(* Logix 5000 project; controller PLC_L27ERM_QBFC1B vendor 1 type 14 code 151 rev 33.13; software revision 33.01 *)

TASK MainTask (continuous, watchdog 500 ms) : MainProgram, CF

MODULES
   Local : vendor 1 type 14 code 151 (Compact 0, rev 33.13)
      Counters : Embedded (Compact 3, rev 1.1, Output RPI 20 ms)
      Discrete_IO : Embedded (Compact 1, rev 3.1, Output RPI 20 ms)
      Analog_IO : Embedded (Compact 2, rev 1.1, Output RPI 80 ms)
      PowerFlex755 : vendor 1 type 143 code 6288 (Ethernet 192.168.2.10, rev 3.2, Output RPI 20 ms)
          : vendor 1 type 143 code 416 (RhinoBP 5, rev 1.8)
          : vendor 1 type 143 code 416 (RhinoBP 4, rev 1.8)
          : vendor 1 type 143 code 32928 (RhinoBP 13, rev 1.1)
          : vendor 1 type 143 code 416 (RhinoBP 6, rev 1.8)
          : vendor 1 type 143 code 33184 (RhinoBP 14, rev 2.5)
END_MODULES

TYPE AnlgIn :
STRUCT
   SCALE_CH : SCALE[4];
   Selector_CH : INT[4];
   PresionEntrada : REAL;
   PresionDescarga : REAL;
   TemperaturaEntrada : REAL;
   TemperaturaDescarga : REAL;
   TemperaturaMotor : REAL;
   PresionCasing : REAL;
   PresionTHP : REAL;
   TemperaturaTHT : REAL;
   ReferenciaAnlg : REAL;
   CTTransformadorElevador : REAL;
   Vibration : REAL;
   CorrienteFuga : REAL;
END_STRUCT
END_TYPE

TYPE DHS :   // Datos sensor de fondo
STRUCT
   PresionEntrada : REAL;
   PresionDescarga : REAL;
   TemperaturaEntrada : REAL;
   TemperaturaDescarga : REAL;
   TemperaturaMotor : REAL;
   PresionCasing : REAL;
   PresionTHP : REAL;
   TemperaturaTHT : REAL;
   Fuente : BOOL;
   Vibration : REAL;
   CorrienteFuga : REAL;
END_STRUCT
END_TYPE

TYPE DInput :   // Fn. Entrada digital
STRUCT
   Start : BMUX;   // Arranque
   Stop : BMUX;   // Parada
   Reset : BMUX;   // Reset
   StopESD : BMUX;   // ESD
   DisparoAltoNivelAceiteSUT : BMUX;   // Disparo SUT
   DisparoAltaTemperaturaSUT : BMUX;   // Disparo SUT
   AlarmaAltaTemperaturaSUT : BMUX;   // Alarma SUT
   AlarmaBajoNivelAceiteSUT : BMUX;   // Alarma SUT
   DisparoBajoBajoNivelAceiteSUT : BMUX;   // Disparo SUT
   DisparoValvulaSobrePresionSUT : BMUX;   // Disparo SUT
   DisparoSobreTensionSUT : BMUX;   // Disparo Tension
   AlarmaDPS : BMUX;   // Alarma DPS
   DisparoAltaTemperaturaFiltros : BMUX;   // Disparo Filtros
   DisparoAltaPresionTHP : BMUX;   // Disparo Instrumentación
   DisparoAltaTemperaturaTHT : BMUX;   // Disparo Instrumentación
   StopESDRemoto : BMUX;   // ESD Remoto
   DisparoPuertaAbierta : BMUX;   // Disparo CILA2S
   DisparoTermicoMotor : BMUX;   // Disparo Motor
   DisparoShutdownSCC : BMUX;   // Disparo SCC
   DisparoBajaPresionTroncal : BMUX;   // Disparo SCC
END_STRUCT
END_TYPE

TYPE DOutput :   // Salida digital
STRUCT
   DO0 : BMUX;
   DO1 : BMUX;
   DO2 : BMUX;
   DO3 : BMUX;
   DO4 : BMUX;
   DO5 : BMUX;
   DO6 : BMUX;
   DO7 : BMUX;
END_STRUCT
END_TYPE

TYPE Filtro :   // Filtro armónicos
STRUCT
   Valor : REAL;
   Referencia : REAL;
   TiempoMuerto : TIMER;
   Output : BOOL;
END_STRUCT
END_TYPE

TYPE IOFn :   // Fn. Salida digital
STRUCT
   DisparoBreakerESD : BOOL;
   FiltroArmonicos : BOOL;
   FallaGeneral : BOOL;
   EstadoCILA2S : BOOL;   // 1:Activo 0:Detenido
   IOFnWord : INT;
END_STRUCT
END_TYPE

ADD_ON_INSTRUCTION BMUX   (* revision 1.1 Multiplexor, vendor Jorge Alberto MartÃ­nez SuÃ¡rez *)
// Multiplexor digital 16:1
// Revision note:
// Se contemplan entradas NO y NC
VAR_INPUT
   Input : INT; {visible}   // Entrada MUX
END_VAR
VAR_OUTPUT
   Output : BOOL; {visible}   // Salida MUX
END_VAR
VAR_INPUT
   Selector : INT; {visible}   // Selector MUX
   Type : BOOL; {visible}
END_VAR

ROUTINE Logic   (* structured text *)
   // Case para las entradas del Add-On
   case Selector of
   	0: 	Output 	:= 0;
   	1: 	Output 	:= Input.0;
   	2: 	Output 	:= Input.1;
   	3: 	Output 	:= Input.2;
   	4: 	Output 	:= Input.3;
   	5: 	Output 	:= Input.4;
   	6: 	Output 	:= Input.5;
   	7: 	Output 	:= Input.6;
   	8: 	Output 	:= Input.7;
   	9: 	Output 	:= Input.8;
   	10: Output 	:= Input.9;
   	11: Output 	:= Input.10;
   	12: Output 	:= Input.11;
   	13: Output 	:= Input.12;
   	14: Output 	:= Input.13;
   	15: Output 	:= Input.14;
   	16: Output	:= Input.15;
   	else
   		Output 	:= 0;
   end_case;
   
   // Tipo de entrada 0:NO 1:NC
   if Type then
   	Output := NOT Output;
   end_if;
   
   // Deshabilitar Salida del Add-On
   if NOT EnableIn then
   	Output := 0;
   end_if;
END_ROUTINE
END_ADD_ON_INSTRUCTION

VAR_GLOBAL   (* controller tags *)
   EstadoDrive : BOOL;
   RelTX : REAL := 1.0;
   Reset : BOOL;
   TensionEntrada : REAL;
END_VAR

PROGRAM CF   (* main routine MainRoutineCF *)
VAR
   AtSetpointSPD : BOOL;
   MtrSpd : REAL;
   PR_E : INT;
   PRDHz : REAL;
   PRH : REAL;
   PRHMS : REAL;
   PRHz : REAL;
   PRM : REAL;
   PRS : REAL;
   RefNotReached : BOOL;
   RefReached : BOOL;
   Rtrn : REAL;
   Start : BOOL;
END_VAR

ROUTINE MainRoutineCF   (* ladder *)
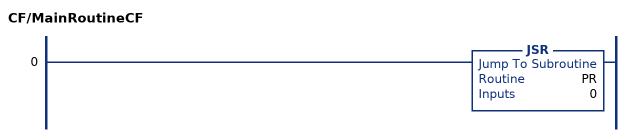
   0: JSR(PR,0);
END_ROUTINE

ROUTINE PR   (* structured text *)
   // LÓGICA SECUENCIAL
   // E0 -> E1
   if PR_E.0 AND Start then
   	PR_E.1:=1; PR_E.0:=0;
   end_if;
   
   // E1 -> E2
   if PR_E.1 AND AtSetpointSPD then
   	PR_E.2:=1; PR_E.1:=0;
   end_if;
   
   // E2 -> E1
   if PR_E.2 AND RefNotReached then
   	PR_E.1:=1; PR_E.2:=0;
   end_if;
   
   // E2 -> E0
   if PR_E.2 AND RefReached then
   	PR_E.0:=1; PR_E.2:=0;
   end_if;
   
   // LÓGICA COMBINACIONAL
   // Estado 0
   if PR_E.0 then
   	PRHMS:= PRH*3600 + PRM*60 + PRS;
   end_if;
   
   // Estado 1
   if PR_E.1 & (PRHz < MtrSpd) then
   	Rtrn := MtrSpd - PRDHz;
   end_if;
   
   if PR_E.1 & (PRHz > MtrSpd) then
   	Rtrn := MtrSpd + PRDHz;
   end_if;
END_ROUTINE
END_PROGRAM

PROGRAM MainProgram   (* main routine MainRoutine *)
VAR
   AnlgFn : AnlgIn;
   CorrienteMotor : REAL;
   DInput : DInput := (Start.Selector := 1, Stop.Selector := 2, Reset.Selector := 3);
   DOutput : DOutput := (DO0.Selector := 4);
   HF : Filtro := (Referencia := 100.0, TiempoMuerto.PRE := 10000);
   index : INT;
   IOFn : IOFn;
        .IOFnWord.0   // Falla general
        .IOFnWord.1   // Disparo breaker ESD
        .IOFnWord.2   // Filtro de armónicos
        .IOFnWord.3   // Estado CILA2S (Activo/Detenido)
   ParadaProteccion : INT;   // Lista de paradas por protección
        .0   // Parada por Presión de entrada
        .1   // Parada por presión de descarga
        .10   // Parada por BUS DC
        .11   // Parada por corriente de salida VSD
        .12   // Parada por tensión de entrada
        .13   // Parada por corriente de motor
        .2   // Parada por temperatura de entrada
        .3   // Parada por temperatura de descarga
        .4   // Parada por temperatura de motor
        .5   // Parada por presión de casing
        .6   // Parada por presión THP
        .7   // Parada por temperatura THT
        .8   // Parada por Vibración
        .9   // Parada por corriente de fuga
   ProtBusDC : ALARM_ANALOG;
   ProtCorrienteFuga : ALARM_ANALOG;
   ProtCorrienteMotor : ALARM_ANALOG;
   ProtOutputCurrent : ALARM_ANALOG;
   ProtPresionCasing : ALARM_ANALOG;
   ProtPresionDescarga : ALARM_ANALOG;
   ProtPresionEntrada : ALARM_ANALOG;
   ProtPresionTHP : ALARM_ANALOG;
   ProtStopVSD : INT;
   ProtTemperaturaDescarga : ALARM_ANALOG;
   ProtTemperaturaEntrada : ALARM_ANALOG;
   ProtTemperaturaMotor : ALARM_ANALOG;
   ProtTemperaturaTHT : ALARM_ANALOG;
   ProtTensionEntrada : ALARM_ANALOG;
   ProtVibration : ALARM_ANALOG;
   SensorFondo : DHS;
END_VAR

ROUTINE AnlgIn   (* structured text *)
   // Escalizar todos los canales
   AnlgFn.SCALE_CH[0].In := Local:2:I.Ch0Data;
   AnlgFn.SCALE_CH[1].In := Local:2:I.Ch1Data;
   AnlgFn.SCALE_CH[2].In := Local:2:I.Ch2Data;
   AnlgFn.SCALE_CH[3].In := Local:2:I.Ch3Data;
   
   // For para asignar las variables de proceso
   for index:=0 to 3 do
   	case AnlgFn.Selector_CH[index] of
   	1: AnlgFn.PresionEntrada := AnlgFn.SCALE_CH[index].Out;
   	2: AnlgFn.PresionDescarga:= AnlgFn.SCALE_CH[index].Out;
   	3: AnlgFn.TemperaturaEntrada := AnlgFn.SCALE_CH[index].Out;
   	4: AnlgFn.TemperaturaDescarga:= AnlgFn.SCALE_CH[index].Out;
   	5: AnlgFn.TemperaturaMotor:= AnlgFn.SCALE_CH[index].Out;
   	6: AnlgFn.PresionCasing:= AnlgFn.SCALE_CH[index].Out;
   	7: AnlgFn.PresionTHP:= AnlgFn.SCALE_CH[index].Out;
   	8: AnlgFn.TemperaturaTHT:= AnlgFn.SCALE_CH[index].Out;
   	9: AnlgFn.ReferenciaAnlg:= AnlgFn.SCALE_CH[index].Out;
   	10: AnlgFn.CTTransformadorElevador:= AnlgFn.SCALE_CH[index].Out;
   	11: AnlgFn.Vibration:= AnlgFn.SCALE_CH[index].Out;
   	12: AnlgFn.CorrienteFuga:= AnlgFn.SCALE_CH[index].Out;
   
   	end_case;
   end_for;
END_ROUTINE

ROUTINE DigitalFn   (* ladder *)
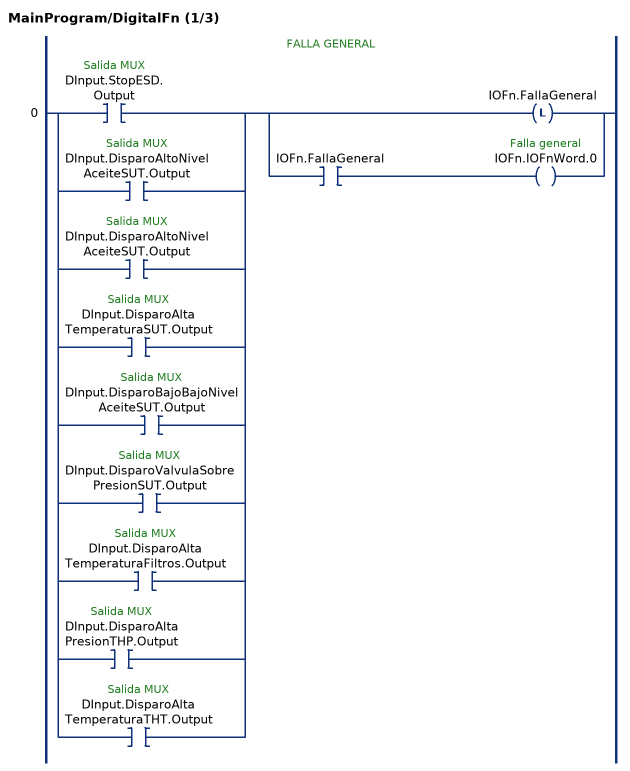
   // FALLA GENERAL
   0: [XIC(DInput.StopESD.Output) ,XIC(DInput.DisparoAltoNivelAceiteSUT.Output) ,XIC(DInput.DisparoAltoNivelAceiteSUT.Output) ,XIC(DInput.DisparoAltaTemperaturaSUT.Output) ,XIC(DInput.DisparoBajoBajoNivelAceiteSUT.Output) ,XIC(DInput.DisparoValvulaSobrePresionSUT.Output) ,XIC(DInput.DisparoAltaTemperaturaFiltros.Output) ,XIC(DInput.DisparoAltaPresionTHP.Output) ,XIC(DInput.DisparoAltaTemperaturaTHT.Output) ][OTL(IOFn.FallaGeneral) ,XIC(IOFn.FallaGeneral) OTE(IOFn.IOFnWord.0) ];
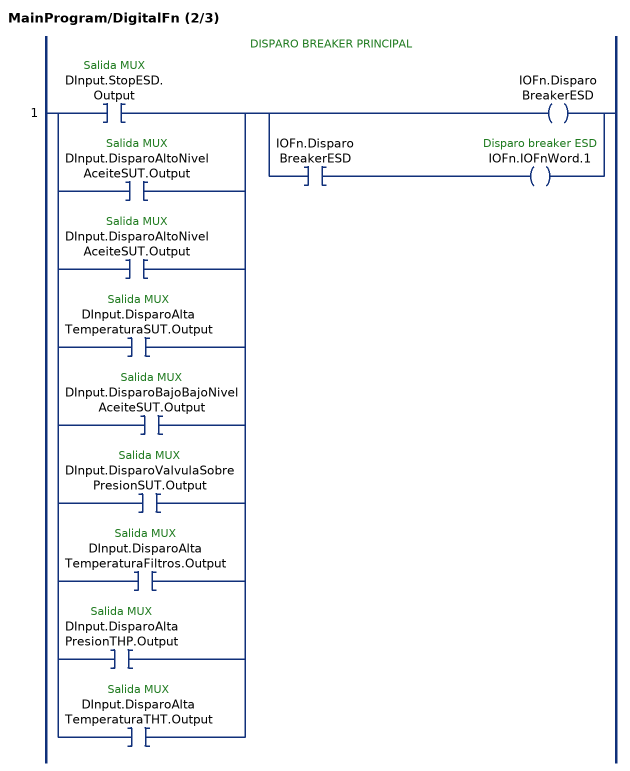
   // DISPARO BREAKER PRINCIPAL
   1: [XIC(DInput.StopESD.Output) ,XIC(DInput.DisparoAltoNivelAceiteSUT.Output) ,XIC(DInput.DisparoAltoNivelAceiteSUT.Output) ,XIC(DInput.DisparoAltaTemperaturaSUT.Output) ,XIC(DInput.DisparoBajoBajoNivelAceiteSUT.Output) ,XIC(DInput.DisparoValvulaSobrePresionSUT.Output) ,XIC(DInput.DisparoAltaTemperaturaFiltros.Output) ,XIC(DInput.DisparoAltaPresionTHP.Output) ,XIC(DInput.DisparoAltaTemperaturaTHT.Output) ][OTE(IOFn.DisparoBreakerESD) ,XIC(IOFn.DisparoBreakerESD) OTE(IOFn.IOFnWord.1) ];
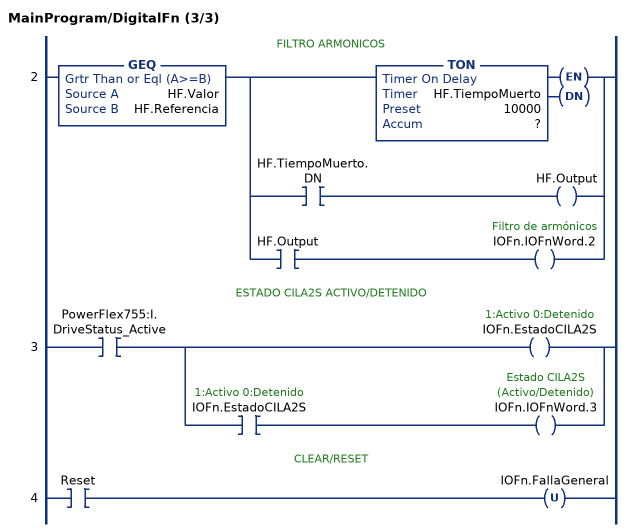
   // FILTRO ARMONICOS
   2: GEQ(HF.Valor,HF.Referencia)[TON(HF.TiempoMuerto,?,?) ,XIC(HF.TiempoMuerto.DN) OTE(HF.Output) ,XIC(HF.Output) OTE(IOFn.IOFnWord.2) ];
   // ESTADO CILA2S ACTIVO/DETENIDO
   3: XIC(PowerFlex755:I.DriveStatus_Active)[OTE(IOFn.EstadoCILA2S) ,XIC(IOFn.EstadoCILA2S) OTE(IOFn.IOFnWord.3) ];
   // CLEAR/RESET
   4: XIC(Reset)OTU(IOFn.FallaGeneral);
END_ROUTINE

ROUTINE InputLD   (* ladder *)
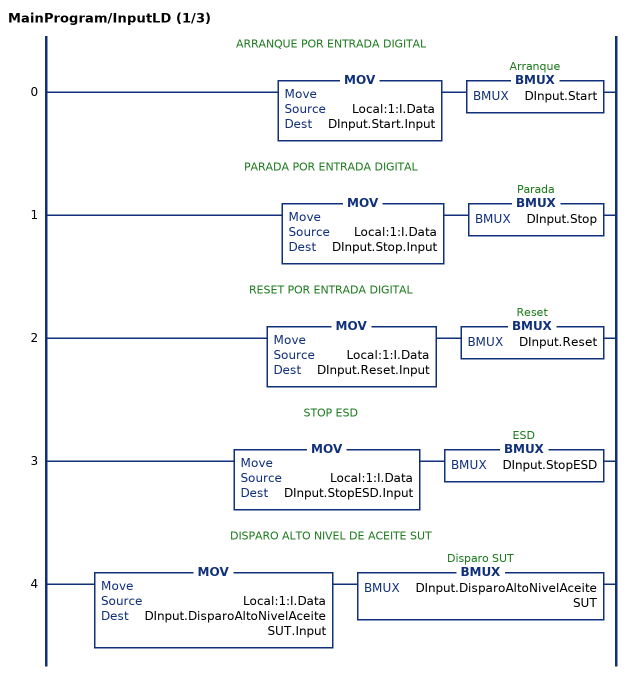
   // ARRANQUE POR ENTRADA DIGITAL
   0: MOV(Local:1:I.Data,DInput.Start.Input)BMUX(DInput.Start);
   // PARADA POR ENTRADA DIGITAL
   1: MOV(Local:1:I.Data,DInput.Stop.Input)BMUX(DInput.Stop);
   // RESET POR ENTRADA DIGITAL
   2: MOV(Local:1:I.Data,DInput.Reset.Input)BMUX(DInput.Reset);
   // STOP ESD
   3: MOV(Local:1:I.Data,DInput.StopESD.Input)BMUX(DInput.StopESD);
   // DISPARO ALTO NIVEL DE ACEITE SUT
   4: MOV(Local:1:I.Data,DInput.DisparoAltoNivelAceiteSUT.Input)BMUX(DInput.DisparoAltoNivelAceiteSUT);
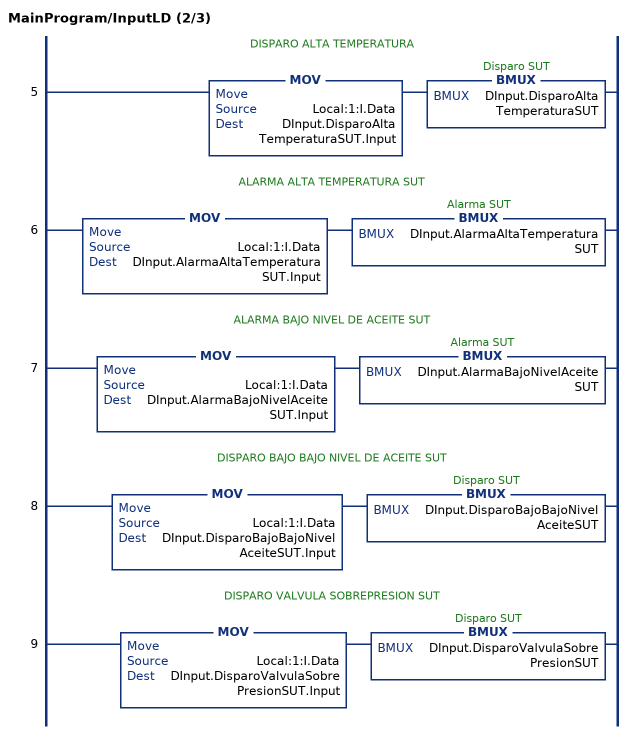
   // DISPARO ALTA TEMPERATURA
   5: MOV(Local:1:I.Data,DInput.DisparoAltaTemperaturaSUT.Input)BMUX(DInput.DisparoAltaTemperaturaSUT);
   // ALARMA ALTA TEMPERATURA SUT
   6: MOV(Local:1:I.Data,DInput.AlarmaAltaTemperaturaSUT.Input)BMUX(DInput.AlarmaAltaTemperaturaSUT);
   // ALARMA BAJO NIVEL DE ACEITE SUT
   7: MOV(Local:1:I.Data,DInput.AlarmaBajoNivelAceiteSUT.Input)BMUX(DInput.AlarmaBajoNivelAceiteSUT);
   // DISPARO BAJO BAJO NIVEL DE ACEITE SUT
   8: MOV(Local:1:I.Data,DInput.DisparoBajoBajoNivelAceiteSUT.Input)BMUX(DInput.DisparoBajoBajoNivelAceiteSUT);
   // DISPARO VALVULA SOBREPRESION SUT
   9: MOV(Local:1:I.Data,DInput.DisparoValvulaSobrePresionSUT.Input)BMUX(DInput.DisparoValvulaSobrePresionSUT);
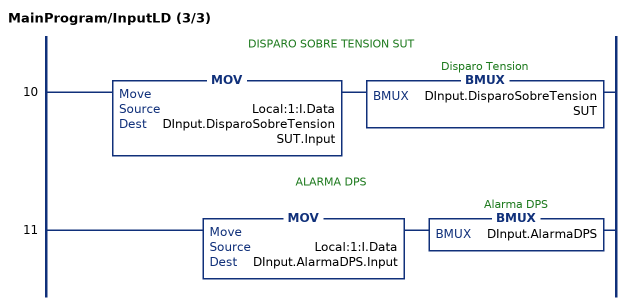
   // DISPARO SOBRE TENSION SUT
   10: MOV(Local:1:I.Data,DInput.DisparoSobreTensionSUT.Input)BMUX(DInput.DisparoSobreTensionSUT);
   // ALARMA DPS
   11: MOV(Local:1:I.Data,DInput.AlarmaDPS.Input)BMUX(DInput.AlarmaDPS);
END_ROUTINE

ROUTINE MainRoutine   (* ladder *)
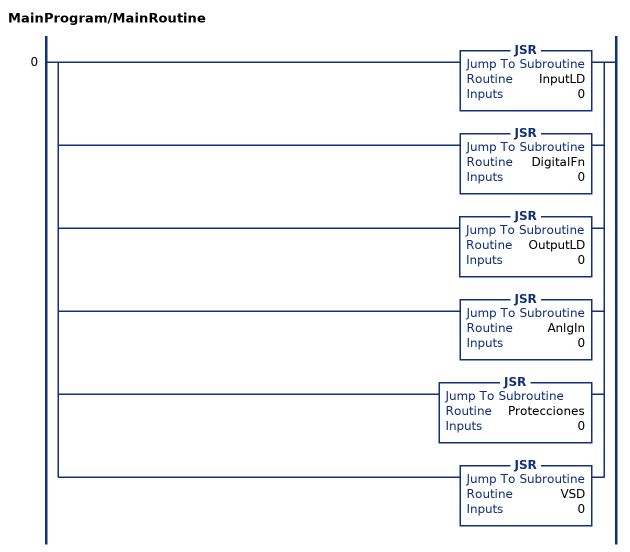
   0: [JSR(InputLD,0) ,JSR(DigitalFn,0) ,JSR(OutputLD,0) ,JSR(AnlgIn,0) ,JSR(Protecciones,0) ,JSR(VSD,0) ];
END_ROUTINE

ROUTINE OutputLD   (* ladder *)
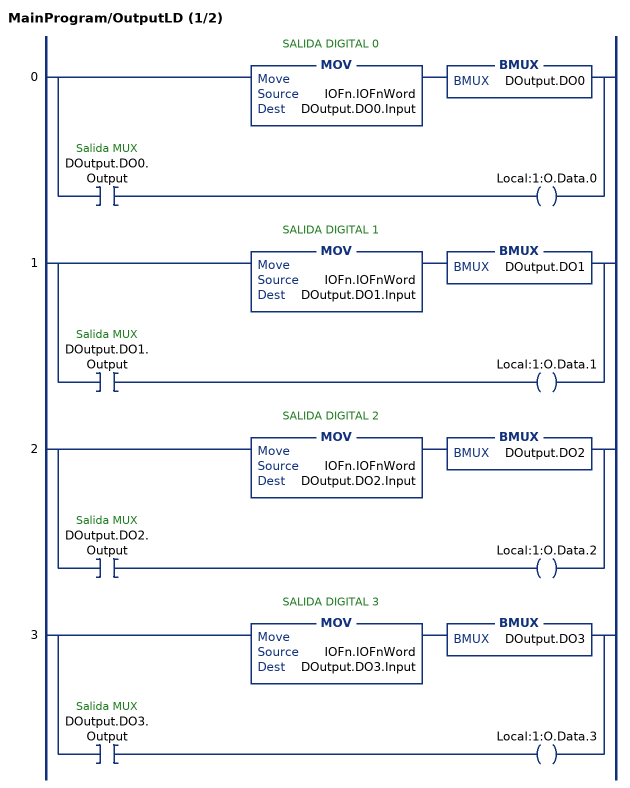
   // SALIDA DIGITAL 0
   0: [MOV(IOFn.IOFnWord,DOutput.DO0.Input) BMUX(DOutput.DO0) ,XIC(DOutput.DO0.Output) OTE(Local:1:O.Data.0) ];
   // SALIDA DIGITAL 1
   1: [MOV(IOFn.IOFnWord,DOutput.DO1.Input) BMUX(DOutput.DO1) ,XIC(DOutput.DO1.Output) OTE(Local:1:O.Data.1) ];
   // SALIDA DIGITAL 2
   2: [MOV(IOFn.IOFnWord,DOutput.DO2.Input) BMUX(DOutput.DO2) ,XIC(DOutput.DO2.Output) OTE(Local:1:O.Data.2) ];
   // SALIDA DIGITAL 3
   3: [MOV(IOFn.IOFnWord,DOutput.DO3.Input) BMUX(DOutput.DO3) ,XIC(DOutput.DO3.Output) OTE(Local:1:O.Data.3) ];
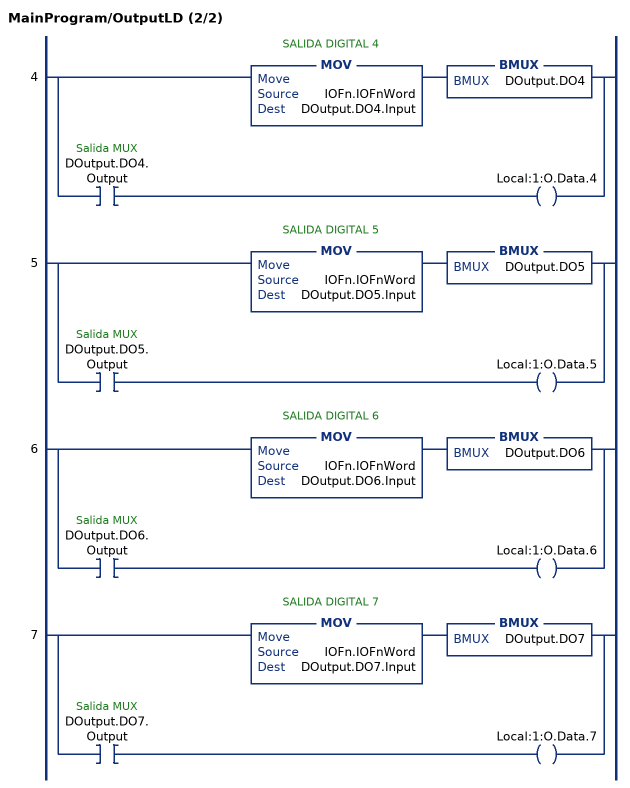
   // SALIDA DIGITAL 4
   4: [MOV(IOFn.IOFnWord,DOutput.DO4.Input) BMUX(DOutput.DO4) ,XIC(DOutput.DO4.Output) OTE(Local:1:O.Data.4) ];
   // SALIDA DIGITAL 5
   5: [MOV(IOFn.IOFnWord,DOutput.DO5.Input) BMUX(DOutput.DO5) ,XIC(DOutput.DO5.Output) OTE(Local:1:O.Data.5) ];
   // SALIDA DIGITAL 6
   6: [MOV(IOFn.IOFnWord,DOutput.DO6.Input) BMUX(DOutput.DO6) ,XIC(DOutput.DO6.Output) OTE(Local:1:O.Data.6) ];
   // SALIDA DIGITAL 7
   7: [MOV(IOFn.IOFnWord,DOutput.DO7.Input) BMUX(DOutput.DO7) ,XIC(DOutput.DO7.Output) OTE(Local:1:O.Data.7) ];
END_ROUTINE

ROUTINE Protecciones   (* ladder *)
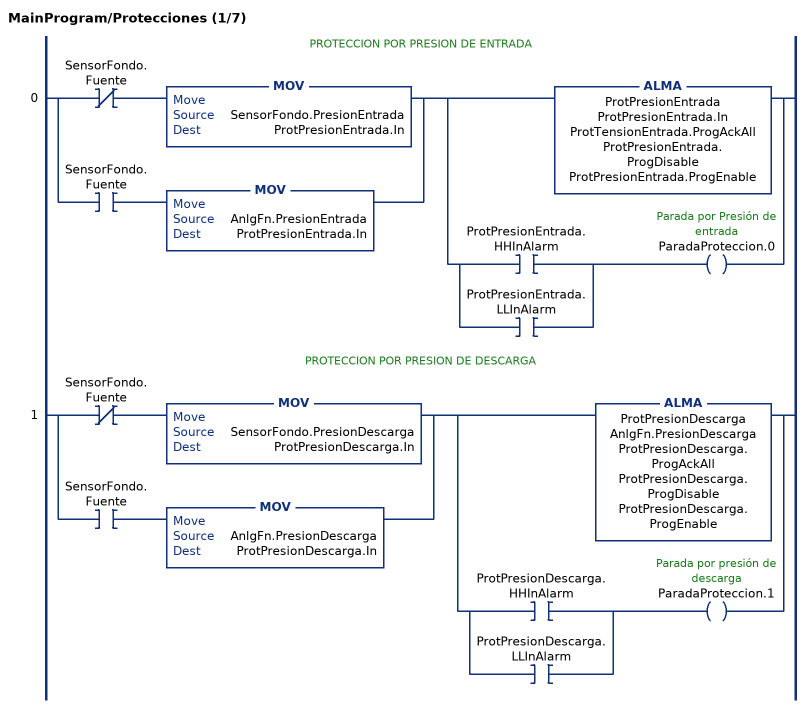
   // PROTECCION POR PRESION DE ENTRADA
   0: [XIO(SensorFondo.Fuente) MOV(SensorFondo.PresionEntrada,ProtPresionEntrada.In) ,XIC(SensorFondo.Fuente) MOV(AnlgFn.PresionEntrada,ProtPresionEntrada.In) ][ALMA(ProtPresionEntrada,ProtPresionEntrada.In,ProtTensionEntrada.ProgAckAll,ProtPresionEntrada.ProgDisable,ProtPresionEntrada.ProgEnable) ,[XIC(ProtPresionEntrada.HHInAlarm) ,XIC(ProtPresionEntrada.LLInAlarm) ] OTE(ParadaProteccion.0) ];
   // PROTECCION POR PRESION DE DESCARGA
   1: [XIO(SensorFondo.Fuente) MOV(SensorFondo.PresionDescarga,ProtPresionDescarga.In) ,XIC(SensorFondo.Fuente) MOV(AnlgFn.PresionDescarga,ProtPresionDescarga.In) ][ALMA(ProtPresionDescarga,AnlgFn.PresionDescarga,ProtPresionDescarga.ProgAckAll,ProtPresionDescarga.ProgDisable,ProtPresionDescarga.ProgEnable) ,[XIC(ProtPresionDescarga.HHInAlarm) ,XIC(ProtPresionDescarga.LLInAlarm) ] OTE(ParadaProteccion.1) ];
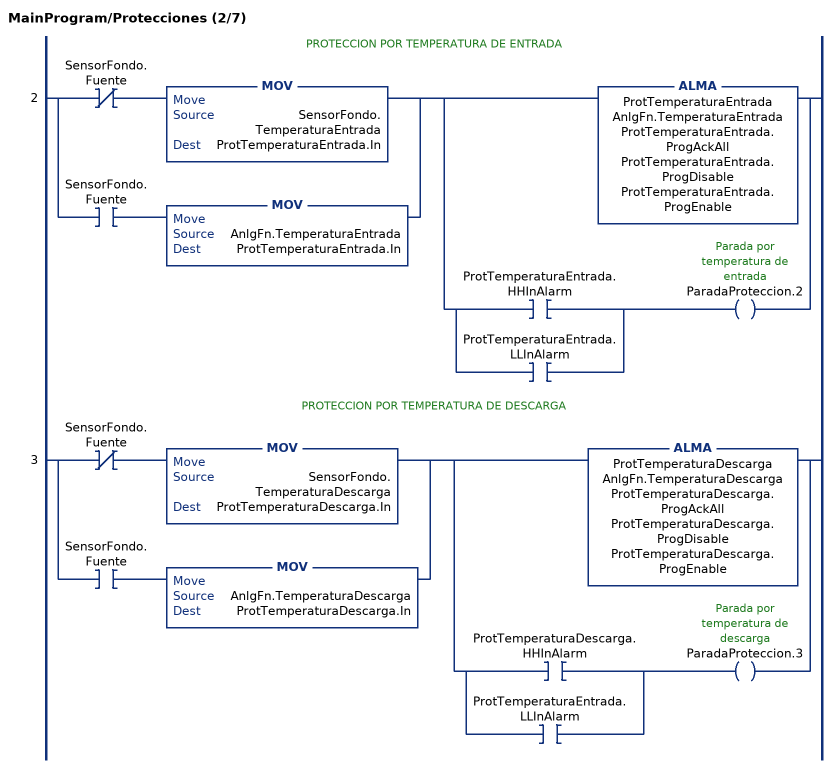
   // PROTECCION POR TEMPERATURA DE ENTRADA
   2: [XIO(SensorFondo.Fuente) MOV(SensorFondo.TemperaturaEntrada,ProtTemperaturaEntrada.In) ,XIC(SensorFondo.Fuente) MOV(AnlgFn.TemperaturaEntrada,ProtTemperaturaEntrada.In) ][ALMA(ProtTemperaturaEntrada,AnlgFn.TemperaturaEntrada,ProtTemperaturaEntrada.ProgAckAll,ProtTemperaturaEntrada.ProgDisable,ProtTemperaturaEntrada.ProgEnable) ,[XIC(ProtTemperaturaEntrada.HHInAlarm) ,XIC(ProtTemperaturaEntrada.LLInAlarm) ] OTE(ParadaProteccion.2) ];
   // PROTECCION POR TEMPERATURA DE DESCARGA
   3: [XIO(SensorFondo.Fuente) MOV(SensorFondo.TemperaturaDescarga,ProtTemperaturaDescarga.In) ,XIC(SensorFondo.Fuente) MOV(AnlgFn.TemperaturaDescarga,ProtTemperaturaDescarga.In) ][ALMA(ProtTemperaturaDescarga,AnlgFn.TemperaturaDescarga,ProtTemperaturaDescarga.ProgAckAll,ProtTemperaturaDescarga.ProgDisable,ProtTemperaturaDescarga.ProgEnable) ,[XIC(ProtTemperaturaDescarga.HHInAlarm) ,XIC(ProtTemperaturaEntrada.LLInAlarm) ] OTE(ParadaProteccion.3) ];
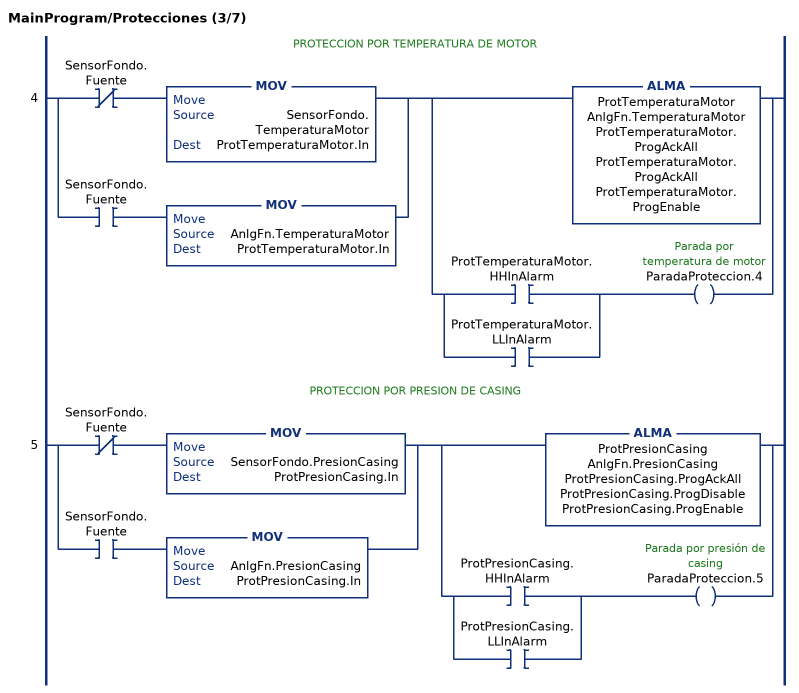
   // PROTECCION POR TEMPERATURA DE MOTOR
   4: [XIO(SensorFondo.Fuente) MOV(SensorFondo.TemperaturaMotor,ProtTemperaturaMotor.In) ,XIC(SensorFondo.Fuente) MOV(AnlgFn.TemperaturaMotor,ProtTemperaturaMotor.In) ][ALMA(ProtTemperaturaMotor,AnlgFn.TemperaturaMotor,ProtTemperaturaMotor.ProgAckAll,ProtTemperaturaMotor.ProgAckAll,ProtTemperaturaMotor.ProgEnable) ,[XIC(ProtTemperaturaMotor.HHInAlarm) ,XIC(ProtTemperaturaMotor.LLInAlarm) ] OTE(ParadaProteccion.4) ];
   // PROTECCION POR PRESION DE CASING
   5: [XIO(SensorFondo.Fuente) MOV(SensorFondo.PresionCasing,ProtPresionCasing.In) ,XIC(SensorFondo.Fuente) MOV(AnlgFn.PresionCasing,ProtPresionCasing.In) ][ALMA(ProtPresionCasing,AnlgFn.PresionCasing,ProtPresionCasing.ProgAckAll,ProtPresionCasing.ProgDisable,ProtPresionCasing.ProgEnable) ,[XIC(ProtPresionCasing.HHInAlarm) ,XIC(ProtPresionCasing.LLInAlarm) ] OTE(ParadaProteccion.5) ];
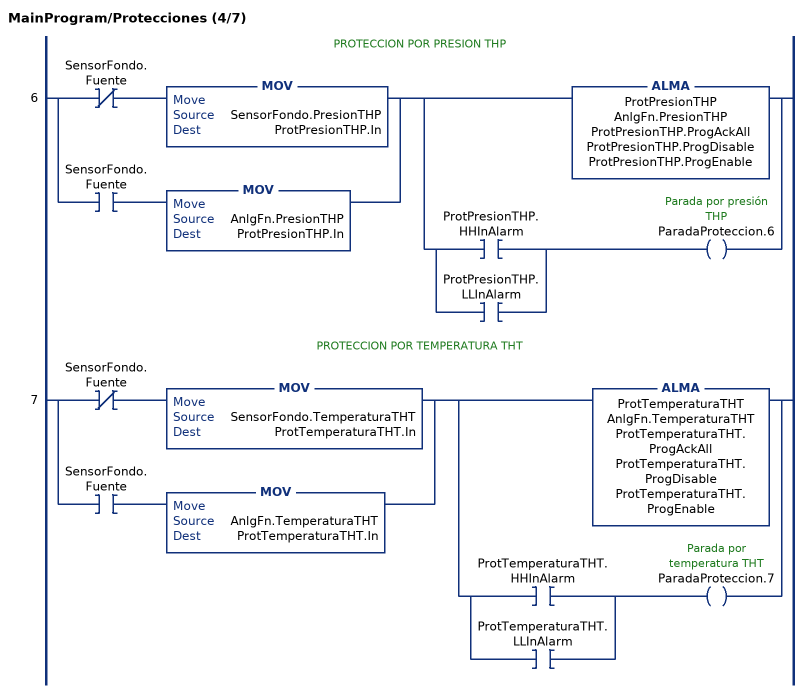
   // PROTECCION POR PRESION THP
   6: [XIO(SensorFondo.Fuente) MOV(SensorFondo.PresionTHP,ProtPresionTHP.In) ,XIC(SensorFondo.Fuente) MOV(AnlgFn.PresionTHP,ProtPresionTHP.In) ][ALMA(ProtPresionTHP,AnlgFn.PresionTHP,ProtPresionTHP.ProgAckAll,ProtPresionTHP.ProgDisable,ProtPresionTHP.ProgEnable) ,[XIC(ProtPresionTHP.HHInAlarm) ,XIC(ProtPresionTHP.LLInAlarm) ] OTE(ParadaProteccion.6) ];
   // PROTECCION POR TEMPERATURA THT
   7: [XIO(SensorFondo.Fuente) MOV(SensorFondo.TemperaturaTHT,ProtTemperaturaTHT.In) ,XIC(SensorFondo.Fuente) MOV(AnlgFn.TemperaturaTHT,ProtTemperaturaTHT.In) ][ALMA(ProtTemperaturaTHT,AnlgFn.TemperaturaTHT,ProtTemperaturaTHT.ProgAckAll,ProtTemperaturaTHT.ProgDisable,ProtTemperaturaTHT.ProgEnable) ,[XIC(ProtTemperaturaTHT.HHInAlarm) ,XIC(ProtTemperaturaTHT.LLInAlarm) ] OTE(ParadaProteccion.7) ];
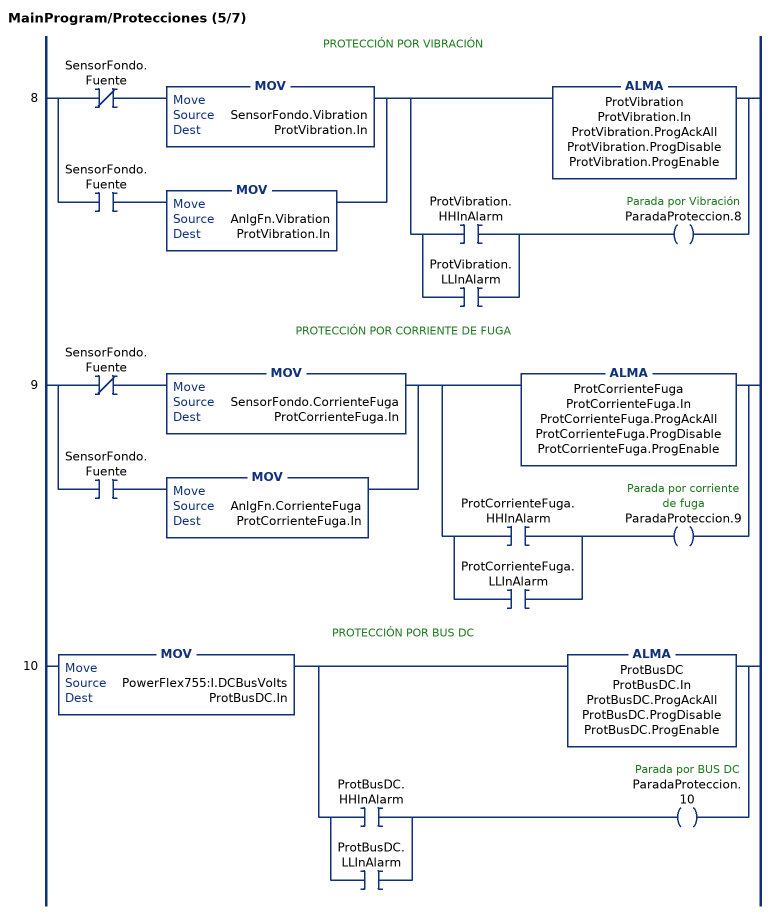
   // PROTECCIÓN POR VIBRACIÓN
   8: [XIO(SensorFondo.Fuente) MOV(SensorFondo.Vibration,ProtVibration.In) ,XIC(SensorFondo.Fuente) MOV(AnlgFn.Vibration,ProtVibration.In) ][ALMA(ProtVibration,ProtVibration.In,ProtVibration.ProgAckAll,ProtVibration.ProgDisable,ProtVibration.ProgEnable) ,[XIC(ProtVibration.HHInAlarm) ,XIC(ProtVibration.LLInAlarm) ] OTE(ParadaProteccion.8) ];
   // PROTECCIÓN POR CORRIENTE DE FUGA
   9: [XIO(SensorFondo.Fuente) MOV(SensorFondo.CorrienteFuga,ProtCorrienteFuga.In) ,XIC(SensorFondo.Fuente) MOV(AnlgFn.CorrienteFuga,ProtCorrienteFuga.In) ][ALMA(ProtCorrienteFuga,ProtCorrienteFuga.In,ProtCorrienteFuga.ProgAckAll,ProtCorrienteFuga.ProgDisable,ProtCorrienteFuga.ProgEnable) ,[XIC(ProtCorrienteFuga.HHInAlarm) ,XIC(ProtCorrienteFuga.LLInAlarm) ] OTE(ParadaProteccion.9) ];
   // PROTECCIÓN POR BUS DC
   10: MOV(PowerFlex755:I.DCBusVolts,ProtBusDC.In)[ALMA(ProtBusDC,ProtBusDC.In,ProtBusDC.ProgAckAll,ProtBusDC.ProgDisable,ProtBusDC.ProgEnable) ,[XIC(ProtBusDC.HHInAlarm) ,XIC(ProtBusDC.LLInAlarm) ] OTE(ParadaProteccion.10) ];
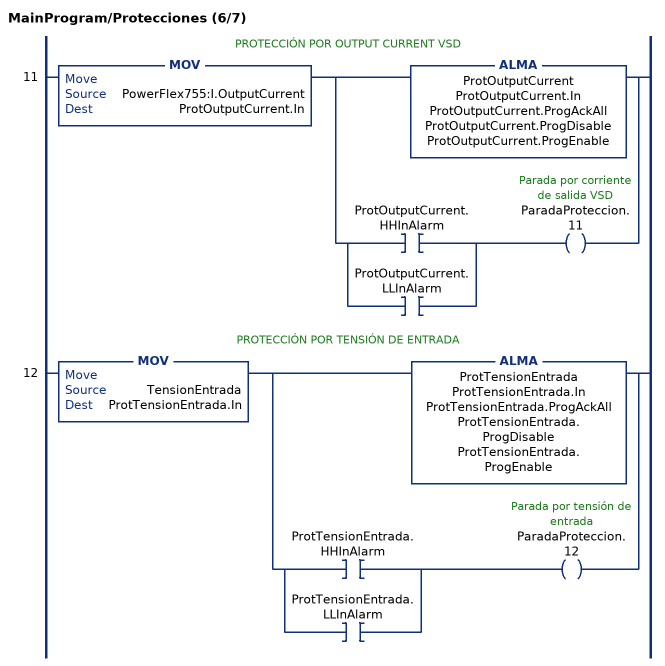
   // PROTECCIÓN POR OUTPUT CURRENT VSD
   11: MOV(PowerFlex755:I.OutputCurrent,ProtOutputCurrent.In)[ALMA(ProtOutputCurrent,ProtOutputCurrent.In,ProtOutputCurrent.ProgAckAll,ProtOutputCurrent.ProgDisable,ProtOutputCurrent.ProgEnable) ,[XIC(ProtOutputCurrent.HHInAlarm) ,XIC(ProtOutputCurrent.LLInAlarm) ] OTE(ParadaProteccion.11) ];
   // PROTECCIÓN POR TENSIÓN DE ENTRADA
   12: MOV(TensionEntrada,ProtTensionEntrada.In)[ALMA(ProtTensionEntrada,ProtTensionEntrada.In,ProtTensionEntrada.ProgAckAll,ProtTensionEntrada.ProgDisable,ProtTensionEntrada.ProgEnable) ,[XIC(ProtTensionEntrada.HHInAlarm) ,XIC(ProtTensionEntrada.LLInAlarm) ] OTE(ParadaProteccion.12) ];
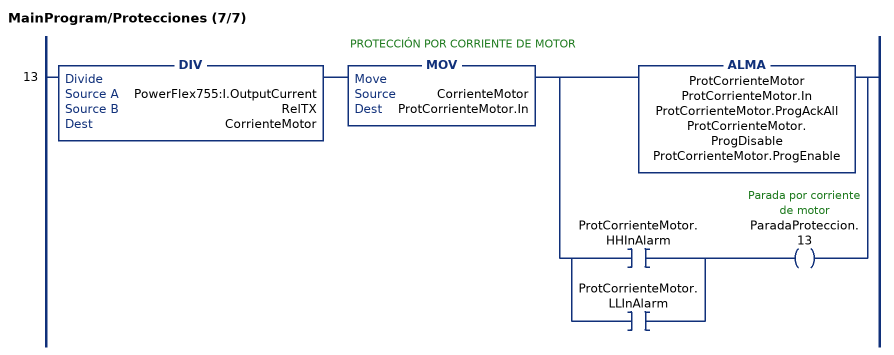
   // PROTECCIÓN POR CORRIENTE DE MOTOR
   13: DIV(PowerFlex755:I.OutputCurrent,RelTX,CorrienteMotor)MOV(CorrienteMotor,ProtCorrienteMotor.In)[ALMA(ProtCorrienteMotor,ProtCorrienteMotor.In,ProtCorrienteMotor.ProgAckAll,ProtCorrienteMotor.ProgDisable,ProtCorrienteMotor.ProgEnable) ,[XIC(ProtCorrienteMotor.HHInAlarm) ,XIC(ProtCorrienteMotor.LLInAlarm) ] OTE(ParadaProteccion.13) ];
END_ROUTINE

ROUTINE VSD   (* ladder *)
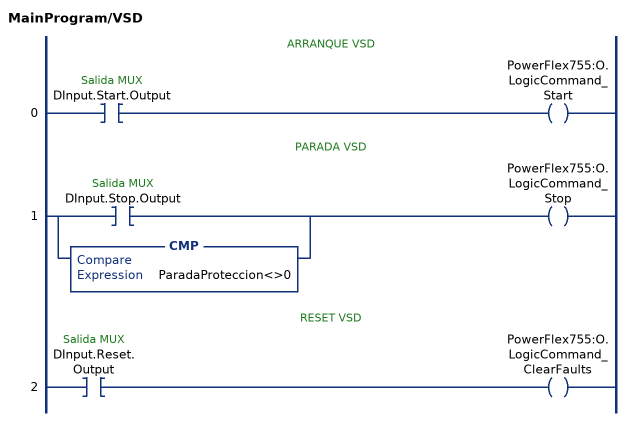
   // ARRANQUE VSD
   0: XIC(DInput.Start.Output)OTE(PowerFlex755:O.LogicCommand_Start);
   // PARADA VSD
   1: [XIC(DInput.Stop.Output) ,CMP(ParadaProteccion<>0) ]OTE(PowerFlex755:O.LogicCommand_Stop);
   // RESET VSD
   2: XIC(DInput.Reset.Output)OTE(PowerFlex755:O.LogicCommand_ClearFaults);
END_ROUTINE
END_PROGRAM
